ABB RobotStudio station: RADomaci22_79_22_175.rspag

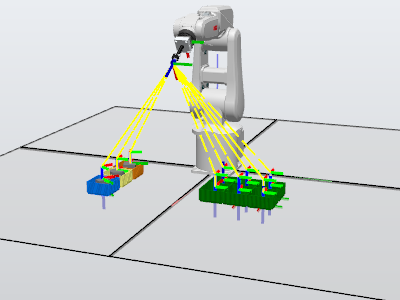
--- station ---
Station RA_Template (saved by RobotStudio 25.3.11371.0)
Controller IRB120_3_58
  mechanical unit ROB_1: IRB120_3_58__01, 6 joints, base frame (0, 0, 0) mm
Layout (positions relative to the parent item):
  - IRB120_3_58__01 [mechanism, from %ABB.RobotStudio.Models.IRB120%\IRB120_3_58_G_01.rslib] at (0, 0, 0) mm; joint values [0, 0, 0, 0, 0.5236, 0] (rad or m)
  - Vakuum_Griepr [mechanism, from Components\Vakuum_Griepr.rslib] at (364.35, 0, 594) mm, rotated rx 180 ry 60 rz 180 deg
  - Box [part] at (219.56, -315.99, 0) mm, size 98.8 x 98.8 x 50 mm
  - Box_2 [part] at (329.12, -315.99, 0) mm, size 98.8 x 98.8 x 50 mm
  - Box_3 [part] at (442.85, -315.99, 0) mm, size 98.8 x 98.8 x 50 mm
  - Box_carier [graphiccomponentgroup] at (55.47, -81.37, 0) mm
    - Box_5 [part] at (219.56, 204.61, -0.53) mm, size 98.8 x 98.8 x 50 mm
    - Box_6 [part] at (219.56, 301.21, 0) mm, size 98.8 x 98.8 x 50 mm
    - Box_7 [part] at (219.56, 395.66, 0) mm, size 98.8 x 98.8 x 50 mm
    - Box_8 [part] at (315.82, 395.66, 0) mm, size 98.8 x 98.8 x 50 mm
    - Box_9 [part] at (315.82, 300.06, 0) mm, size 98.8 x 98.8 x 50 mm
    - Box_10 [part] at (315.82, 205.75, 0) mm, size 98.8 x 98.8 x 50 mm
  - Part_1 [part] at (211.27, -313.8, 52) mm, rotated rx 0 ry 0 rz 20 deg, size 50 x 50 x 50 mm
  - Part_2 [part], size 60 x 60 x 50 mm
  - Part_3 [part] at (444.98, -316.42, 52) mm, rotated rx 0 ry 0 rz -30 deg, size 50 x 30 x 50 mm
Attachment: Vakuum_Griepr is attached to IRB120_3_58__01 / Link6
Attachment: Part_1 is attached to Box
Attachment: Part_2 is attached to Box_2
Attachment: Part_3 is attached to Box_3
Attachment: box1 is attached to Box_5
Attachment: box2 is attached to Box_6
Attachment: box3 is attached to Box_7
Attachment: box4 is attached to Box_8
Attachment: box5 is attached to Box_9
Attachment: box6 is attached to Box_10
Attachment: Workobject_A is attached to Part_1
Attachment: Workobject_B is attached to Part_2
Attachment: Workobject_C is attached to Part_3
Targets, tools, work objects and paths stored in the station and not in the controller backup, written as RAPID:
! task (no controller)
MODULE Module1
  CONST robtarget Target_10:=[[5.789543976,7.220843582,-52],[1,0,0,0],[0,0,0,0],[9E+09,9E+09,9E+09,9E+09,9E+09,9E+09]];
  CONST robtarget Target_10_2:=[[5.789543976,7.220843582,-102],[1,0,0,0],[0,0,0,0],[9E+09,9E+09,9E+09,9E+09,9E+09,9E+09]];
  CONST robtarget Target_20:=[[8.721316961,-2.117156418,-52],[1,0,0,0],[0,0,0,0],[9E+09,9E+09,9E+09,9E+09,9E+09,9E+09]];
  CONST robtarget Target_20_2:=[[8.721316961,-2.117156418,-102],[1,0,0,0],[0,0,0,0],[9E+09,9E+09,9E+09,9E+09,9E+09,9E+09]];
  CONST robtarget Target_30:=[[-2.37647667,-0.382156418,-52],[1,0,0,0],[0,0,0,0],[9E+09,9E+09,9E+09,9E+09,9E+09,9E+09]];
  CONST robtarget Target_30_2:=[[-2.37647667,-0.382156418,-102],[1,0,0,0],[0,0,0,0],[9E+09,9E+09,9E+09,9E+09,9E+09,9E+09]];
ENDMODULE


--- Controller Data/IRB120_3_58/RAPID/TASK1/PROGMOD/CalibData.mod ---
MODULE CalibData
    PERS tooldata Vakuum_Griepr:=[TRUE,[[0,-0.2,130.2],[1,0,0,0]],[0.15,[0,0,52.562],[1,0,0,0],0,0,0]];
    PERS wobjdata box1:=[FALSE,TRUE,"",[[275.029640043,123.239088623,-0.534605694],[1,0,0,0]],[[0,0,50],[1,0,0,0]]];
    PERS wobjdata box2:=[FALSE,TRUE,"",[[275.029640043,219.846654334,0],[1,0,0,0]],[[0,0,0],[0,0,1,0]]];
    PERS wobjdata box3:=[FALSE,TRUE,"",[[275.029640043,314.291802149,0],[0,0,1,0]],[[0,0,0],[1,0,0,0]]];
    PERS wobjdata box4:=[FALSE,TRUE,"",[[371.289668077,314.291802149,0],[1,0,0,0]],[[0,0,0],[0,0,1,0]]];
    PERS wobjdata box5:=[FALSE,TRUE,"",[[371.289668077,218.68993323,0],[1,0,0,0]],[[0,0,0],[0,0,1,0]]];
    PERS wobjdata box6:=[FALSE,TRUE,"",[[371.289668077,124.388795284,0],[0,0,1,0]],[[0,0,0],[1,0,0,0]]];
    PERS wobjdata Workobject_A:=[FALSE,TRUE,"",[[211.268,-310.286390944,52],[0,-0.173648178,0.984807753,0]],[[0,0,0],[1,0,0,0]]];
    PERS wobjdata Workobject_B:=[FALSE,TRUE,"",[[0,0,0],[0,0,1,0]],[[0,0,0],[1,0,0,0]]];
    PERS wobjdata Workobject_C:=[FALSE,TRUE,"",[[444.98260208,-316.417510343,52],[0,0.258819045,0.965925826,0]],[[0,0,50],[1,0,0,0]]];
ENDMODULE

--- Controller Data/IRB120_3_58/RAPID/TASK1/PROGMOD/Module1.mod ---
MODULE Module1
    CONST robtarget Home:=[[477.110403181,-0.2,528.899991815],[0.500000005,0,0.866025401,0],[0,-1,0,0],[9E+09,9E+09,9E+09,9E+09,9E+09,9E+09]];
    VAR robtarget A2:=[[0,0,-50],[1,0,0,0],[-1,0,-1,0],[9E+09,9E+09,9E+09,9E+09,9E+09,9E+09]];
    VAR robtarget A:=[[0,0,0],[1,0,0,0],[-1,0,-1,0],[9E+09,9E+09,9E+09,9E+09,9E+09,9E+09]];
    VAR robtarget B2:=[[-317.402,-318.405,-102],[1,0,0,0],[-1,0,-1,0],[9E+09,9E+09,9E+09,9E+09,9E+09,9E+09]];
    VAR robtarget B:=[[-317.402,-318.405,-52],[1,0,0,0],[-1,0,-1,0],[9E+09,9E+09,9E+09,9E+09,9E+09,9E+09]];
    VAR robtarget C:=[[-2.37647667,-0.382156418,-102],[1,0,0,0],[-1,0,-1,0],[9E+09,9E+09,9E+09,9E+09,9E+09,9E+09]];
    VAR robtarget C_2:=[[-2.37647667,-0.382156418,-52],[1,0,0,0],[-1,0,-1,0],[9E+09,9E+09,9E+09,9E+09,9E+09,9E+09]];
    VAR robtarget Target_40:=[[0,0,50],[0,0,1,0],[0,0,0,0],[9E+09,9E+09,9E+09,9E+09,9E+09,9E+09]];
    VAR robtarget Target_40_2:=[[0,0,0],[0,0,1,0],[0,0,0,0],[9E+09,9E+09,9E+09,9E+09,9E+09,9E+09]];
    VAR robtarget Target_50:=[[0,0,-100],[1,0,0,0],[0,0,0,0],[9E+09,9E+09,9E+09,9E+09,9E+09,9E+09]];
    VAR robtarget Target_50_2:=[[0,0,-50],[1,0,0,0],[0,0,0,0],[9E+09,9E+09,9E+09,9E+09,9E+09,9E+09]];
    VAR robtarget Target_70:=[[0,0,-100],[1,0,0,0],[0,0,0,0],[9E+09,9E+09,9E+09,9E+09,9E+09,9E+09]];
    VAR robtarget Target_70_2:=[[0,0,-50],[1,0,0,0],[0,0,0,0],[9E+09,9E+09,9E+09,9E+09,9E+09,9E+09]];
    VAR robtarget Target_80:=[[0,0,-100],[1,0,0,0],[0,0,0,0],[9E+09,9E+09,9E+09,9E+09,9E+09,9E+09]];
    VAR robtarget Target_80_2:=[[0,0,-50],[1,0,0,0],[0,0,0,0],[9E+09,9E+09,9E+09,9E+09,9E+09,9E+09]];
    VAR robtarget Target_90:=[[0,0,-100],[1,0,0,0],[0,0,0,0],[9E+09,9E+09,9E+09,9E+09,9E+09,9E+09]];
    VAR robtarget Target_90_3:=[[0,0,-50],[1,0,0,0],[0,0,0,0],[9E+09,9E+09,9E+09,9E+09,9E+09,9E+09]];
    VAR robtarget Target_100:=[[0,0,-100],[1,0,0,0],[0,0,0,0],[9E+09,9E+09,9E+09,9E+09,9E+09,9E+09]];
    VAR robtarget Target_100_2:=[[0,0,-50],[1,0,0,0],[0,0,0,0],[9E+09,9E+09,9E+09,9E+09,9E+09,9E+09]];
    !***********************************************************
    !
    ! Module:  Module1
    !
    ! Description:
    !   <Insert description here>
    !
    ! Author: nikolaknezevic
    !
    ! Version: 1.0
    !
    !***********************************************************


    !***********************************************************
    !
    ! Procedure main
    !
    !   This is the entry point of your program
    !
    !***********************************************************
        VAR num brojUredjaja;
        VAR num uredjaji{5};
        VAR num i;
        VAR num id;
        VAR num komponentaA := 0;
        VAR num komponentaB := 0;
        VAR num komponentaC := 0;
        VAR num TMP;
        VAR num brojac := 1;
        VAR robtarget novaMeta;
        VAR num X;
        VAR num Y;
        VAR num teta;
        VAR num seed;

        FUNC robtarget nova_meta(robtarget meta, num X, num Y, num teta)
             novaMeta.trans.x := meta.trans.x + X ;
             novaMeta.trans.y := meta.trans.y + Y ;
             novaMeta.trans.z := meta.trans.z;
             novaMeta.rot := OrientZYX(teta,0,0)*meta.rot;
             novaMeta.robconf := meta.robconf;
             novaMeta.extax := meta.extax;
             RETURN novaMeta;
        ENDFUNC

         PROC kamera(VAR num X , VAR num Y , VAR num teta)
             seed := GetTime(\Msec);

             X := (seed MOD 11) - 5;
             Y := ((seed + 100) MOD 12) - 5;
             teta := ((seed * 2) MOD 13) - 5;
        ENDPROC

    PROC main()
        SetDO Gripper, 0;
        SetDO RobotActive, 0;

        TPReadNum brojUredjaja, "Unesite broj uredjaja (maksimum 5)";
        IF brojUredjaja<1 THEN
            TPWrite("GRESKA! Nema uredjaja za pakovanje.");
            RETURN;
        ELSEIF brojUredjaja>5 THEN
            TPWrite("GRESKA! Unet preveliki broj uredjaja.");
            RETURN;
        ENDIF
        FOR i FROM 1 TO brojUredjaja DO
            TPReadNum uredjaji{i}, "Unesite ID uredjaja (1001,1002,1003,1004):";
            IF (uredjaji{i} > 1004) OR (uredjaji{i} < 1001) THEN
                TPWrite "GRESKA! Unet je nepostojeci ID";
                RETURN;
            ENDIF
        ENDFOR
        FOR i FROM 1 TO brojUredjaja DO
            id := uredjaji{i};
            IF id = 1001 THEN
                komponentaA := komponentaA+1;
                komponentaB := komponentaB+1;
                komponentaC := komponentaC+1;
            ELSEIF id = 1002 THEN
                komponentaA := komponentaA+2;
                komponentaC := komponentaC+1;
            ELSEIF id = 1003 THEN
                komponentaA := komponentaA+2;
                komponentaB := komponentaB+2;
                komponentaC := komponentaC+2;
            ELSEIF id = 1004 THEN
                komponentaA := komponentaA+3;
            ENDIF
        ENDFOR

        IF (komponentaA>10) OR (komponentaB>10) OR (komponentaC>10) THEN
            TPWrite "GRESKA! Potrebno je vise komponenti nego sto je dostupno";
            RETURN;
        ENDIF

        TPWrite "Sve je spremno za rad.";
        TPReadFK TMP, "Da li zapocinjem pakovanje?", "DA","","","","NE";
        IF TMP = 1 THEN
            ! ovde ide celo izvrsavanje
            FOR i FROM 1 TO brojUredjaja DO
                id := uredjaji{i};
                SetDO RobotActive,1;

                IF i = 1 THEN
                    ! postavljanje novih koordinata kutije-nosaca
                    kamera X, Y, teta;

                    Target_40 := nova_meta(Target_40, X , Y , teta);
                    Target_40_2 := nova_meta(Target_40_2, X , Y , teta);
                    Target_50 := nova_meta(Target_50, X , Y , teta);
                    Target_50_2 := nova_meta(Target_50_2, X , Y , teta);
                    Target_70 := nova_meta(Target_70, X , Y , teta);
                    Target_70_2 := nova_meta(Target_70_2, X , Y , teta);
                    Target_80 := nova_meta(Target_80, X , Y , teta);
                    Target_80_2 := nova_meta(Target_80_2, X , Y , teta);
                    Target_90 := nova_meta(Target_90, X , Y , teta);
                    Target_90_3 := nova_meta(Target_90_3, X , Y , teta);
                    Target_100 := nova_meta(Target_100, X , Y , teta);
                    Target_100_2 := nova_meta(Target_100_2, X , Y , teta);
                ENDIF

                IF id = 1001 THEN
                    IF brojac = 1 THEN
                        Home_A;
                        HomeBox1;
                        Home_B;
                        HomeBox2;
                        Home_C;
                        HomeBox3;
                        brojac := 4;
                        IF i = brojUredjaja THEN
                            SetDO RobotActive,0;
                            TPWrite("Poslate su sve komponente. Zadatak je zavrsen.");
                            RETURN;    ! moze da ostane, ispravno
                        ELSEIF uredjaji{i+1} = 1003 THEN
                            brojac := 1;
                            SetDO RobotActive,0;
                            TPWrite("Sledeci uredjaj je prevelik. Zamenite kutiju sada.");
                            TPReadFK TMP, "Da li da nastavim pakovanje?", "DA","","","","NE";
                            IF TMP = 5 THEN
                                TPWrite("Korisnik je prekinuo izvrsavanje programa.");
                                RETURN;
                            ENDIF
                            WHILE TMP <> 1 DO
                                TPReadFK TMP, "Da li da nastavim pakovanje?", "DA","","","","NE";
                            ENDWHILE
                            SetDO RobotActive,1;
                            ! postavljanje novih koordinata kutije-nosaca
                            kamera X, Y, teta;

                            Target_40 := nova_meta(Target_40, X , Y , teta);
                            Target_40_2 := nova_meta(Target_40_2, X , Y , teta);
                            Target_50 := nova_meta(Target_50, X , Y , teta);
                            Target_50_2 := nova_meta(Target_50_2, X , Y , teta);
                            Target_70 := nova_meta(Target_70, X , Y , teta);
                            Target_70_2 := nova_meta(Target_70_2, X , Y , teta);
                            Target_80 := nova_meta(Target_80, X , Y , teta);
                            Target_80_2 := nova_meta(Target_80_2, X , Y , teta);
                            Target_90 := nova_meta(Target_90, X , Y , teta);
                            Target_90_3 := nova_meta(Target_90_3, X , Y , teta);
                            Target_100 := nova_meta(Target_100, X , Y , teta);
                            Target_100_2 := nova_meta(Target_100_2, X , Y , teta);
                        ENDIF
                    ELSEIF brojac = 4 THEN
                        Home_A;
                        HomeBox4;
                        Home_B;
                        HomeBox5;
                        Home_C;
                        HomeBox6;
                        brojac := 1;
                        IF i = brojUredjaja THEN
                            SetDO RobotActive,0;
                            TPWrite("Poslate su sve komponente. Zadatak je zavrsen.");
                            RETURN;
                        ELSE
                            SetDO RobotActive,0;
                            TPWrite("Kutija je puna. Zamenite kutiju sada.");
                            TPReadFK TMP, "Da li da nastavim pakovanje?", "DA","","","","NE";
                            IF TMP = 5 THEN
                                TPWrite("Korisnik je prekinuo izvrsavanje programa.");
                                RETURN;
                            ENDIF
                            WHILE TMP <> 1 DO
                                TPReadFK TMP, "Da li da nastavim pakovanje?", "DA","","","","NE";
                            ENDWHILE
                            SetDO RobotActive,1;
                            ! postavljanje novih koordinata kutije-nosaca
                            kamera X, Y, teta;

                            Target_40 := nova_meta(Target_40, X , Y , teta);
                            Target_40_2 := nova_meta(Target_40_2, X , Y , teta);
                            Target_50 := nova_meta(Target_50, X , Y , teta);
                            Target_50_2 := nova_meta(Target_50_2, X , Y , teta);
                            Target_70 := nova_meta(Target_70, X , Y , teta);
                            Target_70_2 := nova_meta(Target_70_2, X , Y , teta);
                            Target_80 := nova_meta(Target_80, X , Y , teta);
                            Target_80_2 := nova_meta(Target_80_2, X , Y , teta);
                            Target_90 := nova_meta(Target_90, X , Y , teta);
                            Target_90_3 := nova_meta(Target_90_3, X , Y , teta);
                            Target_100 := nova_meta(Target_100, X , Y , teta);
                            Target_100_2 := nova_meta(Target_100_2, X , Y , teta);
                        ENDIF
                    ENDIF

                ELSEIF id = 1002 THEN
                    IF brojac = 1 THEN
                        Home_A;
                        HomeBox1;
                        Home_A;
                        HomeBox2;
                        Home_C;
                        HomeBox3;
                        brojac := 4;
                        IF i = brojUredjaja THEN
                            SetDO RobotActive,0;
                            TPWrite("Poslate su sve komponente. Zadatak je zavrsen.");
                            RETURN;
                        ELSEIF uredjaji{i+1} = 1003 THEN
                            brojac := 1;
                            SetDO RobotActive,0;
                            TPWrite("Sledeci uredjaj je prevelik. Zamenite kutiju sada.");
                            TPReadFK TMP, "Da li da nastavim pakovanje?", "DA","","","","NE";
                            IF TMP = 5 THEN
                                TPWrite("Korisnik je prekinuo izvrsavanje programa.");
                                RETURN;
                            ENDIF
                            WHILE TMP <> 1 DO
                                TPReadFK TMP, "Da li da nastavim pakovanje?", "DA","","","","NE";
                            ENDWHILE
                            SetDO RobotActive,1;
                            kamera X, Y, teta;

                            Target_40 := nova_meta(Target_40, X , Y , teta);
                            Target_40_2 := nova_meta(Target_40_2, X , Y , teta);
                            Target_50 := nova_meta(Target_50, X , Y , teta);
                            Target_50_2 := nova_meta(Target_50_2, X , Y , teta);
                            Target_70 := nova_meta(Target_70, X , Y , teta);
                            Target_70_2 := nova_meta(Target_70_2, X , Y , teta);
                            Target_80 := nova_meta(Target_80, X , Y , teta);
                            Target_80_2 := nova_meta(Target_80_2, X , Y , teta);
                            Target_90 := nova_meta(Target_90, X , Y , teta);
                            Target_90_3 := nova_meta(Target_90_3, X , Y , teta);
                            Target_100 := nova_meta(Target_100, X , Y , teta);
                            Target_100_2 := nova_meta(Target_100_2, X , Y , teta);
                        ENDIF
                    ELSEIF brojac = 4 THEN
                        Home_A;
                        HomeBox4;
                        Home_A;
                        HomeBox5;
                        Home_C;
                        HomeBox6;
                        brojac := 1;
                        IF i = brojUredjaja THEN
                            SetDO RobotActive,0;
                            TPWrite("Poslate su sve komponente. Zadatak je zavrsen.");
                            RETURN;
                        ELSE
                            SetDO RobotActive,0;
                            TPWrite("Kutija je puna. Zamenite kutiju sada.");
                            TPReadFK TMP, "Da li da nastavim pakovanje?", "DA","","","","NE";
                            IF TMP = 5 THEN
                                TPWrite("Korisnik je prekinuo izvrsavanje programa.");
                                RETURN;
                            ENDIF
                            WHILE TMP <> 1 DO
                                TPReadFK TMP, "Da li da nastavim pakovanje?", "DA","","","","NE";
                            ENDWHILE
                            SetDO RobotActive,1;
                            kamera X, Y, teta;

                            Target_40 := nova_meta(Target_40, X , Y , teta);
                            Target_40_2 := nova_meta(Target_40_2, X , Y , teta);
                            Target_50 := nova_meta(Target_50, X , Y , teta);
                            Target_50_2 := nova_meta(Target_50_2, X , Y , teta);
                            Target_70 := nova_meta(Target_70, X , Y , teta);
                            Target_70_2 := nova_meta(Target_70_2, X , Y , teta);
                            Target_80 := nova_meta(Target_80, X , Y , teta);
                            Target_80_2 := nova_meta(Target_80_2, X , Y , teta);
                            Target_90 := nova_meta(Target_90, X , Y , teta);
                            Target_90_3 := nova_meta(Target_90_3, X , Y , teta);
                            Target_100 := nova_meta(Target_100, X , Y , teta);
                            Target_100_2 := nova_meta(Target_100_2, X , Y , teta);
                        ENDIF
                    ENDIF

                ELSEIF id = 1004 THEN
                    IF brojac = 1 THEN
                        Home_A;
                        HomeBox1;
                        Home_A;
                        HomeBox2;
                        Home_A;
                        HomeBox3;
                        brojac := 4;
                        IF i = brojUredjaja THEN
                            SetDO RobotActive,0;
                            TPWrite("Poslate su sve komponente. Zadatak je zavrsen.");
                            RETURN;
                        ELSEIF uredjaji{i+1} = 1003 THEN
                            brojac := 1;
                            SetDO RobotActive,0;
                            TPWrite("Sledeci uredjaj je prevelik. Zamenite kutiju sada.");
                            TPReadFK TMP, "Da li da nastavim pakovanje?", "DA","","","","NE";
                            IF TMP = 5 THEN
                                TPWrite("Korisnik je prekinuo izvrsavanje programa.");
                                RETURN;
                            ENDIF
                            WHILE TMP <> 1 DO
                                TPReadFK TMP, "Da li da nastavim pakovanje?", "DA","","","","NE";
                            ENDWHILE
                            SetDO RobotActive,1;
                            kamera X, Y, teta;

                            Target_40 := nova_meta(Target_40, X , Y , teta);
                            Target_40_2 := nova_meta(Target_40_2, X , Y , teta);
                            Target_50 := nova_meta(Target_50, X , Y , teta);
                            Target_50_2 := nova_meta(Target_50_2, X , Y , teta);
                            Target_70 := nova_meta(Target_70, X , Y , teta);
                            Target_70_2 := nova_meta(Target_70_2, X , Y , teta);
                            Target_80 := nova_meta(Target_80, X , Y , teta);
                            Target_80_2 := nova_meta(Target_80_2, X , Y , teta);
                            Target_90 := nova_meta(Target_90, X , Y , teta);
                            Target_90_3 := nova_meta(Target_90_3, X , Y , teta);
                            Target_100 := nova_meta(Target_100, X , Y , teta);
                            Target_100_2 := nova_meta(Target_100_2, X , Y , teta);
                        ENDIF
                    ELSEIF brojac = 4 THEN
                        Home_A;
                        HomeBox4;
                        Home_A;
                        HomeBox5;
                        Home_A;
                        HomeBox6;
                        brojac := 1;
                        IF i = brojUredjaja THEN
                            SetDO RobotActive,0;
                            TPWrite("Poslate su sve komponente. Zadatak je zavrsen.");
                            RETURN;
                        ELSE
                            SetDO RobotActive,0;
                            TPWrite("Kutija je puna. Zamenite kutiju sada.");
                            TPReadFK TMP, "Da li da nastavim pakovanje?", "DA","","","","NE";
                            IF TMP = 5 THEN
                                TPWrite("Korisnik je prekinuo izvrsavanje programa.");
                                RETURN;
                            ENDIF
                            WHILE TMP <> 1 DO
                                TPReadFK TMP, "Da li da nastavim pakovanje?", "DA","","","","NE";
                            ENDWHILE
                            SetDO RobotActive,1;
                            kamera X, Y, teta;

                            Target_40 := nova_meta(Target_40, X , Y , teta);
                            Target_40_2 := nova_meta(Target_40_2, X , Y , teta);
                            Target_50 := nova_meta(Target_50, X , Y , teta);
                            Target_50_2 := nova_meta(Target_50_2, X , Y , teta);
                            Target_70 := nova_meta(Target_70, X , Y , teta);
                            Target_70_2 := nova_meta(Target_70_2, X , Y , teta);
                            Target_80 := nova_meta(Target_80, X , Y , teta);
                            Target_80_2 := nova_meta(Target_80_2, X , Y , teta);
                            Target_90 := nova_meta(Target_90, X , Y , teta);
                            Target_90_3 := nova_meta(Target_90_3, X , Y , teta);
                            Target_100 := nova_meta(Target_100, X , Y , teta);
                            Target_100_2 := nova_meta(Target_100_2, X , Y , teta);
                        ENDIF
                    ENDIF

                ELSEIF id = 1003 THEN
                    Home_A;
                    HomeBox1;
                    Home_A;
                    HomeBox2;
                    Home_B;
                    HomeBox3;
                    Home_B;
                    HomeBox4;
                    Home_C;
                    HomeBox5;
                    Home_C;
                    HomeBox6;
                    IF i = brojUredjaja THEN
                        SetDO RobotActive,0;
                        TPWrite("Poslate su sve komponente. Zadatak je zavrsen.");
                        RETURN;
                    ELSE
                        SetDO RobotActive,0;
                        TPWrite("Kutija je puna. Zamenite kutiju sada.");
                        TPReadFK TMP, "Da li da nastavim pakovanje?", "DA","","","","NE";
                        IF TMP = 5 THEN
                            TPWrite("Korisnik je prekinuo izvrsavanje programa.");
                            RETURN;
                        ENDIF
                        WHILE TMP <> 1 DO
                            TPReadFK TMP, "Da li da nastavim pakovanje?", "DA","","","","NE";
                        ENDWHILE
                        SetDO RobotActive,1;
                        kamera X, Y, teta;

                        Target_40 := nova_meta(Target_40, X , Y , teta);
                        Target_40_2 := nova_meta(Target_40_2, X , Y , teta);
                        Target_50 := nova_meta(Target_50, X , Y , teta);
                        Target_50_2 := nova_meta(Target_50_2, X , Y , teta);
                        Target_70 := nova_meta(Target_70, X , Y , teta);
                        Target_70_2 := nova_meta(Target_70_2, X , Y , teta);
                        Target_80 := nova_meta(Target_80, X , Y , teta);
                        Target_80_2 := nova_meta(Target_80_2, X , Y , teta);
                        Target_90 := nova_meta(Target_90, X , Y , teta);
                        Target_90_3 := nova_meta(Target_90_3, X , Y , teta);
                        Target_100 := nova_meta(Target_100, X , Y , teta);
                        Target_100_2 := nova_meta(Target_100_2, X , Y , teta);
                    ENDIF
                ENDIF
            ENDFOR
ENDIF
    ENDPROC



    PROC Home_A()
        kamera X, Y, teta;

        A := nova_meta(A, X , Y , teta);
        A2 := nova_meta(A2, X , Y , teta);

        MoveJ Home,v500,fine,Vakuum_Griepr\WObj:=wobj0;
        MoveJ A2,v500,fine,Vakuum_Griepr\WObj:=Workobject_A;
        MoveL A,v100,fine,Vakuum_Griepr\WObj:=Workobject_A;
        WaitTime \InPos, 0.01;
        SetDO Gripper, 1;
        WaitTime 0.5;
        MoveL A2,v100,fine,Vakuum_Griepr\WObj:=Workobject_A;
        MoveJ Home,v500,fine,Vakuum_Griepr\WObj:=wobj0;
    ENDPROC
    PROC Home_B()
        kamera X, Y, teta;

        B := nova_meta(B, X , Y , teta);
        B2 := nova_meta(B2, X , Y , teta);

        MoveJ Home,v500,fine,Vakuum_Griepr\WObj:=wobj0;
        MoveJ B2,v500,fine,Vakuum_Griepr\WObj:=Workobject_B;
        MoveL B,v100,fine,Vakuum_Griepr\WObj:=Workobject_B;
        WaitTime \InPos, 0.01;
        SetDO Gripper, 1;
        WaitTime 0.5;
        MoveL B2,v100,fine,Vakuum_Griepr\WObj:=Workobject_B;
        MoveJ Home,v500,fine,Vakuum_Griepr\WObj:=wobj0;
    ENDPROC
    PROC Home_C()
        kamera X, Y, teta;

        C := nova_meta(C, X , Y , teta);
        C_2 := nova_meta(C_2, X , Y , teta);

        MoveJ Home,v500,fine,Vakuum_Griepr\WObj:=wobj0;
        MoveJ C,v500,fine,Vakuum_Griepr\WObj:=Workobject_C;
        MoveL C_2,v100,fine,Vakuum_Griepr\WObj:=Workobject_C;
        WaitTime \InPos, 0.01;
        SetDO Gripper, 1;
        WaitTime 0.5;
        MoveL C,v100,fine,Vakuum_Griepr\WObj:=Workobject_C;
        MoveJ Home,v500,fine,Vakuum_Griepr\WObj:=wobj0;
    ENDPROC
    PROC HomeBox1()
        MoveJ Home,v500,fine,Vakuum_Griepr\WObj:=wobj0;
        MoveJ Target_40,v500,fine,Vakuum_Griepr\WObj:=box1;
        MoveL Target_40_2,v100,fine,Vakuum_Griepr\WObj:=box1;
        WaitTime \InPos, 0.01;
        SetDO Gripper, 0;
        WaitTime 0.5;
        MoveL Target_40,v100,fine,Vakuum_Griepr\WObj:=box1;
        MoveJ Home,v500,fine,Vakuum_Griepr\WObj:=wobj0;
    ENDPROC
    PROC HomeBox2()
        MoveJ Home,v500,fine,Vakuum_Griepr\WObj:=wobj0;
        MoveJ Target_50,v500,fine,Vakuum_Griepr\WObj:=box2;
        MoveL Target_50_2,v100,fine,Vakuum_Griepr\WObj:=box2;
        WaitTime \InPos, 0.01;
        SetDO Gripper, 0;
        WaitTime 0.5;
        MoveL Target_50,v100,fine,Vakuum_Griepr\WObj:=box2;
        MoveJ Home,v500,fine,Vakuum_Griepr\WObj:=wobj0;
    ENDPROC
    PROC HomeBox3()
        MoveJ Home,v500,fine,Vakuum_Griepr\WObj:=wobj0;
        MoveJ Target_70,v500,fine,Vakuum_Griepr\WObj:=box3;
        MoveL Target_70_2,v100,fine,Vakuum_Griepr\WObj:=box3;
        WaitTime \InPos, 0.01;
        SetDO Gripper, 0;
        WaitTime 0.5;
        MoveL Target_70,v100,fine,Vakuum_Griepr\WObj:=box3;
        MoveJ Home,v500,fine,Vakuum_Griepr\WObj:=wobj0;
    ENDPROC
    PROC HomeBox4()
        MoveJ Home,v500,fine,Vakuum_Griepr\WObj:=wobj0;
        MoveJ Target_80,v500,fine,Vakuum_Griepr\WObj:=box4;
        MoveL Target_80_2,v100,fine,Vakuum_Griepr\WObj:=box4;
        WaitTime \InPos, 0.01;
        SetDO Gripper, 0;
        WaitTime 0.5;
        MoveL Target_80,v100,fine,Vakuum_Griepr\WObj:=box4;
        MoveJ Home,v500,fine,Vakuum_Griepr\WObj:=wobj0;
    ENDPROC
    PROC HomeBox5()
        MoveJ Home,v500,fine,Vakuum_Griepr\WObj:=wobj0;
        MoveJ Target_90,v500,fine,Vakuum_Griepr\WObj:=box5;
        MoveL Target_90_3,v100,fine,Vakuum_Griepr\WObj:=box5;
        WaitTime \InPos, 0.01;
        SetDO Gripper, 0;
        WaitTime 0.5;
        MoveL Target_90,v100,fine,Vakuum_Griepr\WObj:=box5;
        MoveJ Home,v500,fine,Vakuum_Griepr\WObj:=wobj0;
    ENDPROC
    PROC HomeBox6()
        MoveJ Home,v500,fine,Vakuum_Griepr\WObj:=wobj0;
        MoveJ Target_100,v500,fine,Vakuum_Griepr\WObj:=box6;
        MoveL Target_100_2,v100,fine,Vakuum_Griepr\WObj:=box6;
        WaitTime \InPos, 0.01;
        SetDO Gripper, 0;
        WaitTime 0.5;
        MoveL Target_100,v100,fine,Vakuum_Griepr\WObj:=box6;
        MoveJ Home,v500,fine,Vakuum_Griepr\WObj:=wobj0;
    ENDPROC
ENDMODULE

--- Controller Data/IRB120_3_58/SYSPAR/EIO.cfg ---
EIO:CFG_1.0:6:1::
#
EIO_SIGNAL:

      -Name "Gripper" -SignalType "DO" -Access "All"

      -Name "RobotActive" -SignalType "DO" -Access "All"
